Fanuc KAREL source: kd00063.KL

-- PROVISIONAL review KL for V770-1; original PC SHA256 7091271553c3c12d31dc27afdbe446f0b0bcd23e2b547350b357cd3403d119eb
-- Incomplete behavior may be omitted. Consult companion uncertainty JSON. Do not deploy.
PROGRAM KD00063
%NOLOCKGROUP
VAR
  I : INTEGER
  J : INTEGER
  B : BOOLEAN
  R : REAL
  S : STRING[80]
BEGIN
  -- UNRESOLVED_PC offsets 5-18; opcodes 9D,81,18,9D,1B,9D,12,9D,13,04
  -- UNRESOLVED_PC offsets 23-27; opcodes 7F
END KD00063
